Staubli VAL3: cycle_end.pgx

program cycle_end()
begin
  if !cycleStatus:bToEnd and cycleStatus:bCycle
    logMsg("[KERNEL] PLC:End cycle")
    call OnEvent:endCycle()
  endIf
end
